TYPE U_APP_STATE :
UNION
  stState             : ST_APP_STATE;
  byState   AT %i*    : ARRAY[1..SIZEOF(ST_APP_STATE)] OF BYTE;
END_UNION
END_TYPE

(* stored: Version 1.1.0.1
   DUT U_APP_STATE: Id {adcc4659-3bbd-4ee4-ad3a-61625ba0f7fc} *)
